PROGRAM P_2PickUP
VAR
	nState: INT;
	
	//Vision Color for Lid
	Blue:	INT:=3;
	Green:	INT:=6;
	Metal:	INT:=9;
	
	//Timers for the different state to happen. It is good to put in timers so the machinery have time to do the different
	// state before it moves on to the next state else everything will happen really fast.
	fbTimerMoving : TON;	// Timer in the moving state so the XYZ arm have time to process before moving till next state.
	fbTimerPickUP : TON;	 // 
	fbTimerGrab : TON;
	fbTimerGrab2 : TON;
	fbTimerDrop : TON;
	fbTimerMovingLid : TON;
	fbTimerWaiting : TON;
END_VAR

VAR CONSTANT
	//This is the Constant Variables that we use to for the different state in our Case OF Statement.
	Standby: 		INT:=00;
	Start:			INT:=01;
	ReadVision: 	INT:=02;
	atEntry: 		INT:=10;
	Moving: 		INT:=20;
	PickUP:			INT:=21;
	PickUP2: 		INT:=22;
	Grab: 			INT:=23;
	Grab2: 			INT:=24;
	Drop: 			INT:=25;
	MovingLid: 		INT:=26;
	MovingLid2: 	INT:=27;
	MovingStop: 	INT:=29;
	Waiting: 		INT:=30;
	Stopping: 		INT:=40;
	Resetting: 		INT:=50;
	Estop:			INT:=99;
END_VAR

// This is our second program where we emit a base and let the vision cam tell us which color the base is so the first XYZ arm can pick up the lid and send if 
// to pack.


CASE nState OF 
	Standby:	
		IF FIO.bEbStart=TRUE THEN
			nState:=Start;
		END_IF	
	
	Start: 
			IF FIO.bInPaSensBlue AND FIO.bInPaSensGreen AND FIO.bInPaSensMetal THEN
				FIO.bInEmitBase:=TRUE;
				nState:=ReadVision;
			END_IF	
			
	ReadVision: //vision cam read the color of the base
				IF FIO.iInVision=Blue THEN
					FIO.rInPaMoveX:=9;			
					nState:=Moving;	
				END_IF
				IF FIO.iInVision=Green THEN
					FIO.rInPaMoveX:=5;					
					nState:=Moving;
				END_IF
				IF FIO.iInVision=Metal THEN 
					FIO.rInPaMoveX:=1;			
					nState:=Moving;
				END_IF
				
	Moving:
		IF FIO.rInPaMoveX=9 OR FIO.rInPaMoveX=5 OR FIO.rInPaMoveX=1 THEN
			FIO.rInPaMoveY:=0.5;
		 fbTimerMoving(IN:=TRUE,PT:=T#1S);
		 IF fbTimerMoving.Q THEN
			fbTimerMoving(IN:=FALSE);
			nState:=PickUP; 
		 END_IF		
		END_IF
	
	PickUP:
		IF FIO.rInPaMoveY=0.5 THEN
			FIO.rInPaMoveZ:=9;
			FIO.bInPaToolRot:=TRUE;
			fbTimerPickUP(IN:=TRUE,PT:=T#1S);
		 IF fbTimerPickUP.Q THEN
			 fbTimerPickUP(IN:=FALSE);
			nState:=Grab; 
		 END_IF	
		END_IF
		
	Grab:
		IF FIO.rInPaMoveZ=9 THEN
			FIO.bInPaGrab:=TRUE;
		fbTimerGrab(IN:=TRUE,PT:=T#1S);
		 IF fbTimerGrab.Q THEN
			fbTimerGrab(IN:=FALSE);
			nState:=Grab2; 
		 END_IF
		END_IF
		
	Grab2:	
		IF FIO.bInPaGrab=TRUE THEN
			FIO.rInPaMoveZ:=5;
			FIO.rInPaMoveY:=8;
			fbTimerGrab2(IN:=TRUE,PT:=T#1S);	
			IF fbTimerGrab2.Q THEN
				fbTimerGrab2(IN:=FALSE);
				nState:=Drop;
		 	END_IF				
		END_IF
	
	Drop:
		IF FIO.bInPaGrab=TRUE THEN
			FIO.rInPaMoveZ:=8.5;
			fbTimerDrop(IN:=TRUE,PT:=T#1S);	
			IF fbTimerDrop.Q THEN
				fbTimerDrop(IN:=FALSE);
				nState:=MovingLid; 
		 	END_IF
		 END_IF
		 
	MovingLid:				
			IF FIO.rInPaMoveZ=8.5 THEN
				FIO.bInPaGrab:=FALSE;
			END_IF
				fbTimerMovingLid(IN:=TRUE,PT:=T#1S);	
			IF fbTimerMovingLid.Q THEN
				fbTimerMovingLid(IN:=FALSE);
				nState:=MovingLid2; 
		 	END_IF
			
	MovingLid2:		
			IF FIO.bInPaGrab=FALSE THEN
				FIO.rInPaMoveX:=0;
				FIO.rInPaMoveY:=0;
				FIO.rInPaMoveZ:=0;
				FIO.bInPaToolRot:=FALSE;
				FIO.bInConvSorting:=TRUE;
				nState:=waiting; 	
			END_IF
//----------------------------------------------------------------------------//
	Waiting:
			IF FIO.bPP_LidClamp=TRUE THEN
			fbTimerWaiting(IN:=TRUE,PT:=T#1S);	
			IF fbTimerWaiting.Q THEN
				fbTimerWaiting(IN:=FALSE); 
				nState:=Start;
			END_IF
			END_IF
//----------------------------------------------------------------------------//

		

	
	Stopping:
		IF FIO.bEbStop = FALSE THEN
			FIO.bEbStopLight:=TRUE;
		ELSIF FIO.bEbReset=TRUE THEN
				FIO.bEbStopLight:=FALSE;	
			nState:=Standby;	
		END_IF	

//----------------------------------------------------------------------------// 
	ELSE
		nState:=9999;	
END_CASE

IF NOT FIO.bEbStop THEN
		nState:=Stopping;	
END_IF

END_PROGRAM

(* stored: Version 1.1.0.1, ProductVersion 3.1.4024.3
   POU P_2PickUP: Id {f81accdf-79ad-420e-a6ed-ebdb2655ce8e}, SpecialFunc None *)
